// TIA Portal project "factoryIO_from_a2b" (V19)

(* hardware
DEVICE "S7-1200 station_1"  S7-1200 Station
   slot 0: "Rack_0"  S7-1200 Rack  Rack  V1.0
   slot 1: "PLC_1"  CPU 1212C DC/DC/Rly  6ES7 212-1HE40-0XB0  V4.5
*)

// ===== PLC "PLC_1"  CPU 1212C DC/DC/Rly =====

VAR_GLOBAL   // PLC tag table "Default tag table"
   "Start" AT %I10.0 : Bool;
   "Conveyor" AT %Q0.0 : Bool;
   "Sensor" AT %I0.1 : Bool;
END_VAR

ORGANIZATION_BLOCK "Main"   // OB1, LAD, ProgramCycle
TITLE = "Main Program Sweep (Cycle)"
{ S7_Optimized_Access := 'TRUE' }
VERSION : 0.1
   VAR_INPUT
      Initial_Call : Bool;   // Initial call of this OB
      Remanence : Bool;   // =True, if remanent data are available
   END_VAR
BEGIN

REGION Network 1
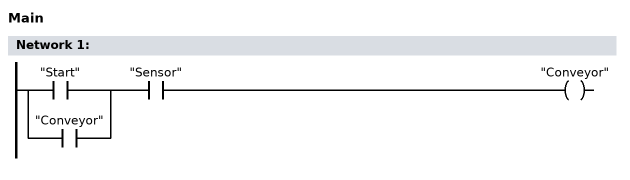
   RUNG wire#powerrail
      Contact( "Start" )
      wire#w1
      Contact( "Sensor" )
      Coil( "Conveyor" )
   END_RUNG
   RUNG wire#powerrail
      Contact( "Conveyor" )
   END_RUNG wire#w1
   // the same network as SCL:
   "Conveyor" := ("Start" OR "Conveyor") AND "Sensor";
END_REGION
END_ORGANIZATION_BLOCK